# EPICS substitutions: app/Db/tpr_master.substitutions
file tpr_config.template
{
pattern {  IOC    }
        { $(IOC) }
}

file tpr_ch_config.template
{
pattern { N, L,     RATE,      FLSTAT   ,  FHSTAT }
        { 0, 1, 8.403361345, "INVALID"  , "INVALID"},
        { 1, 1, 8.403361345, "INVALID"  , "INVALID"},
        { 2, 1, 8.403361345, "INVALID"  , "INVALID"},
        { 3, 1, 8.403361345, "INVALID"  , "INVALID"},
        { 4, 1, 8.403361345, "INVALID"  , "INVALID"},
        { 5, 1, 8.403361345, "INVALID"  , "INVALID"},
        { 6, 1, 8.403361345, "INVALID"  , "INVALID"},
        { 7, 1, 8.403361345, "INVALID"  , "INVALID"},
        { 8, 1, 8.403361345, "INVALID"  , "INVALID"},
        { 9, 1, 8.403361345, "INVALID"  , "INVALID"},
        { A, 1, 8.403361345, "INVALID"  , "INVALID"},
        { B, 1, 8.403361345, "INVALID"  , "INVALID"},
        { 0, 2, 5.385029618, "NO_ALARM" , "MAJOR" },
        { 1, 2, 5.385029618, "NO_ALARM" , "MAJOR" },
        { 2, 2, 5.385029618, "NO_ALARM" , "MAJOR" },
        { 3, 2, 5.385029618, "NO_ALARM" , "MAJOR" },
        { 4, 2, 5.385029618, "NO_ALARM" , "MAJOR" },
        { 5, 2, 5.385029618, "NO_ALARM" , "MAJOR" },
        { 6, 2, 5.385029618, "NO_ALARM" , "MAJOR" },
        { 7, 2, 5.385029618, "NO_ALARM" , "MAJOR" },
        { 8, 2, 5.385029618, "NO_ALARM" , "MAJOR" },
        { 9, 2, 5.385029618, "NO_ALARM" , "MAJOR" },
        { A, 2, 5.385029618, "NO_ALARM" , "MAJOR" },
        { B, 2, 5.385029618, "NO_ALARM", "MAJOR"  }
}
